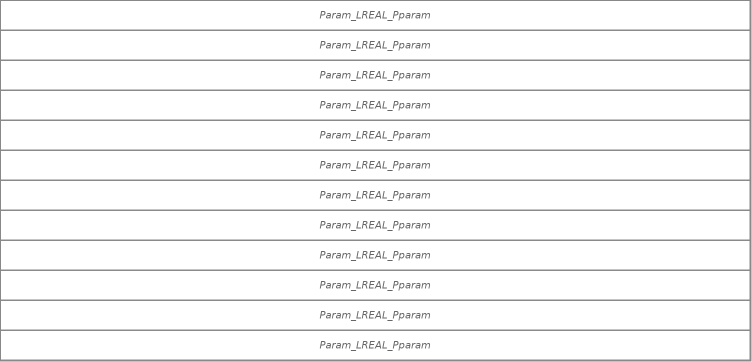
VISUALIZATION Visu_PParam_Params  // 752x362
    Frame (0,0 750x30)
        shows Param_LREAL_Pparam(nIdx := GlobalOne)
    Frame (0,30 750x30)
        shows Param_LREAL_Pparam(nIdx := 2)
    Frame (0,60 750x30)
        shows Param_LREAL_Pparam(nIdx := 3)
    Frame (0,90 750x30)
        shows Param_LREAL_Pparam(nIdx := 4)
    Frame (0,120 750x30)
        shows Param_LREAL_Pparam(nIdx := 5)
    Frame (0,150 750x30)
        shows Param_LREAL_Pparam(nIdx := 6)
    Frame (0,180 750x30)
        shows Param_LREAL_Pparam(nIdx := 7)
    Frame (0,210 750x30)
        shows Param_LREAL_Pparam(nIdx := 8)
    Frame (0,240 750x30)
        shows Param_LREAL_Pparam(nIdx := 9)
    Frame (0,270 750x30)
        shows Param_LREAL_Pparam(nIdx := 10)
    Frame (0,300 750x30)
        shows Param_LREAL_Pparam(nIdx := 11)
    Frame (0,330 750x30)
        shows Param_LREAL_Pparam(nIdx := 12)
END_VISUALIZATION

(* stored: Version 1.1.0.1
   Visu Visu_PParam_Params: Id {69fe28ba-fecf-4e23-a85b-52f1be8fcd78} *)
